INTERFACE I_MachineControl EXTENDS I_UniversalMachine

PROPERTY Robots : REFERENCE TO FB_Robot
GET
END_GET
END_PROPERTY

PROPERTY StateInit : REFERENCE TO E_MachineCtrlStateInit
GET
END_GET
END_PROPERTY

PROPERTY StateUninitialized : REFERENCE TO E_MachineCtrlStateUninitialized
GET
END_GET
END_PROPERTY

END_INTERFACE

(* stored: Version 1.1.0.1, ProductVersion 3.1.4024.9
   Itf I_MachineControl: Id {575cfd35-d864-4f94-b2bb-e1e7c6df6ebc}
   Property Robots: Id {508a7188-8eec-4c0a-b26d-0bdcd24ff2fb}
   Get Get: Id {eed6073b-58a6-4232-ab65-7b3da114e4ea}
   Property StateInit: Id {2aa14ad1-e093-419a-baca-f8ea9fb7ba74}
   Get Get: Id {9c85bcf2-b125-47be-bfc2-fdec58190f47}
   Property StateUninitialized: Id {509c677d-4d2e-47b1-9d76-81dd936053aa}
   Get Get: Id {262865c9-dfe6-451e-bad3-c65870effd61} *)
